// Mitsubishi GX Works2 project: PLC SAMPLE Conveyor   PLC: Q00J

PROGRAM MAIN
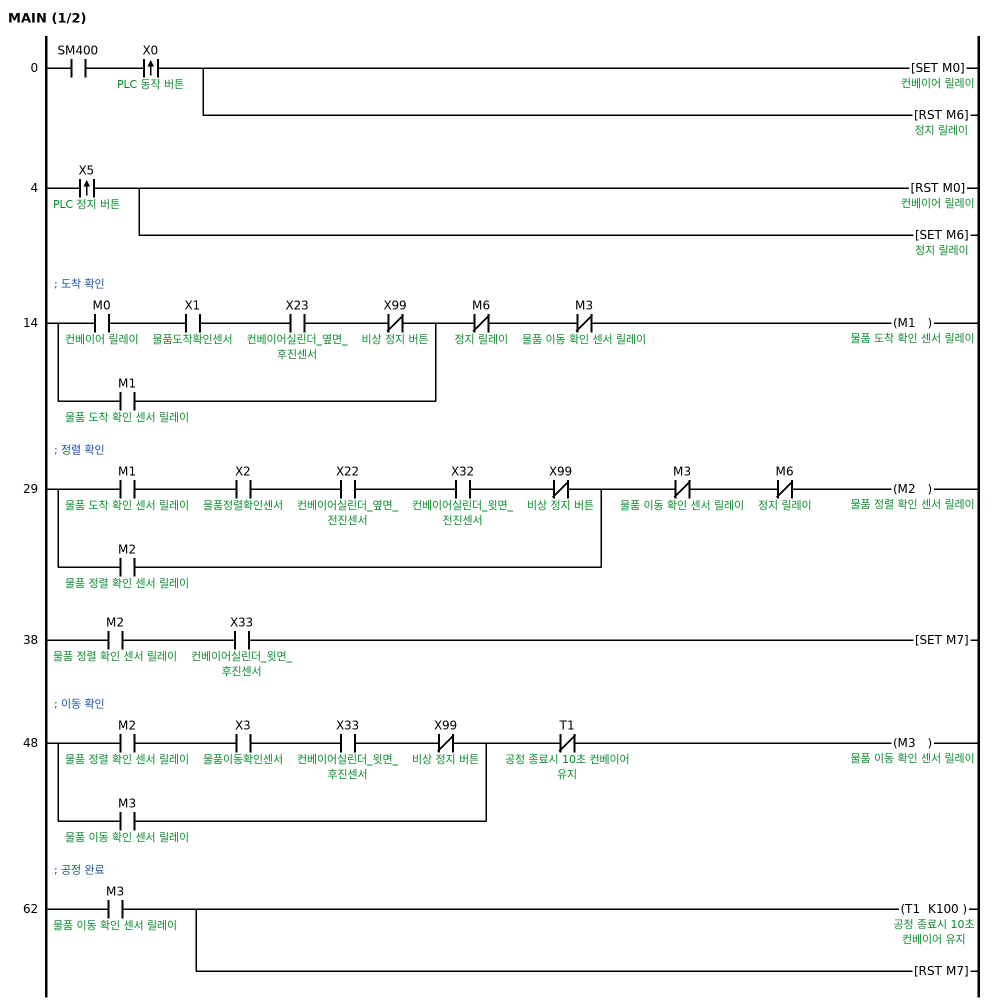
0     LD      SM400
      ANDP    X0  ; PLC 동작 버튼
      SET     M0  ; 컨베이어 릴레이
      RST     M6  ; 정지 릴레이
4     LDP     X5  ; PLC 정지 버튼
      RST     M0  ; 컨베이어 릴레이
      SET     M6  ; 정지 릴레이
; 도착 확인
14    LD      M0  ; 컨베이어 릴레이
      AND     X1  ; 물품도착확인센서
      AND     X23  ; 컨베이어실린더_옆면_후진센서
      ANI     X99  ; 비상 정지 버튼
      OR      M1  ; 물품 도착 확인 센서 릴레이
      ANI     M6  ; 정지 릴레이
      ANI     M3  ; 물품 이동 확인 센서 릴레이
      OUT     M1  ; 물품 도착 확인 센서 릴레이
; 정렬 확인
29    LD      M1  ; 물품 도착 확인 센서 릴레이
      AND     X2  ; 물품정렬확인센서
      AND     X22  ; 컨베이어실린더_옆면_전진센서
      AND     X32  ; 컨베이어실린더_윗면_전진센서
      ANI     X99  ; 비상 정지 버튼
      OR      M2  ; 물품 정렬 확인 센서 릴레이
      ANI     M3  ; 물품 이동 확인 센서 릴레이
      ANI     M6  ; 정지 릴레이
      OUT     M2  ; 물품 정렬 확인 센서 릴레이
38    LD      M2  ; 물품 정렬 확인 센서 릴레이
      AND     X33  ; 컨베이어실린더_윗면_후진센서
      SET     M7
; 이동 확인
48    LD      M2  ; 물품 정렬 확인 센서 릴레이
      AND     X3  ; 물품이동확인센서
      AND     X33  ; 컨베이어실린더_윗면_후진센서
      ANI     X99  ; 비상 정지 버튼
      OR      M3  ; 물품 이동 확인 센서 릴레이
      ANI     T1  ; 공정 종료시 10초 컨베이어 유지
      OUT     M3  ; 물품 이동 확인 센서 릴레이
; 공정 완료
62    LD      M3  ; 물품 이동 확인 센서 릴레이
      OUT     T1 K100  ; 공정 종료시 10초 컨베이어 유지
      RST     M7
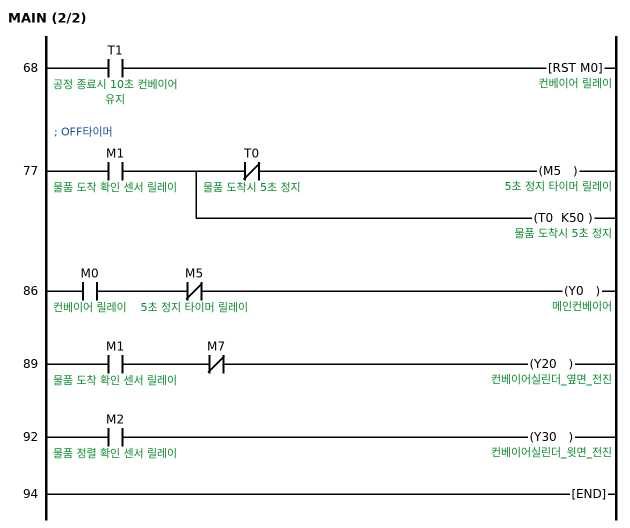
68    LD      T1  ; 공정 종료시 10초 컨베이어 유지
      RST     M0  ; 컨베이어 릴레이
; OFF타이머
77    LD      M1  ; 물품 도착 확인 센서 릴레이
      MPS
      ANI     T0  ; 물품 도착시 5초 정지
      OUT     M5  ; 5초 정지 타이머 릴레이
      MPP
      OUT     T0 K50  ; 물품 도착시 5초 정지
86    LD      M0  ; 컨베이어 릴레이
      ANI     M5  ; 5초 정지 타이머 릴레이
      OUT     Y0  ; 메인컨베이어
89    LD      M1  ; 물품 도착 확인 센서 릴레이
      ANI     M7
      OUT     Y20  ; 컨베이어실린더_옆면_전진
92    LD      M2  ; 물품 정렬 확인 센서 릴레이
      OUT     Y30  ; 컨베이어실린더_윗면_전진
94    END
END_PROGRAM
